PROGRAM Cabinet_Monitoring
VAR
    //fbCabinetMonitoring: FB_ESSMonitoringMCU5001a; FB_ESSMonitoringMCU5001b; FB_ESSMonitoringMCU6001a; FB_ESSMonitoringMCU6001b; FB_ESSMonitoringMCU5002; FB_ESSMonitoringMCU5003;
END_VAR

//Cabinet monitoring
//fbCabinetMonitoring(
//    nEcMasterNetId := '10.102.116.36.3.1', //AMS NetId of Device (EtherCAT) from I/Os,
//    iSafetyProvider := Motion_Safety.fbMotionSafety,
//    aErrorID => ,
//    aErrorMsg => ,
//    nEcMasterFramesLost => ,
//    nCPULoad => ,
//    fCycleExecTime_ms => ,
//    nAlarmGrpBitNumber =>
//);

END_PROGRAM

(* stored: Version 1.1.0.1
   POU Cabinet_Monitoring: Id {f09ddf2c-38c8-0b17-348a-c2e3aa836c88}, SpecialFunc None *)
